ABB RAPID module: offs_inline.mod

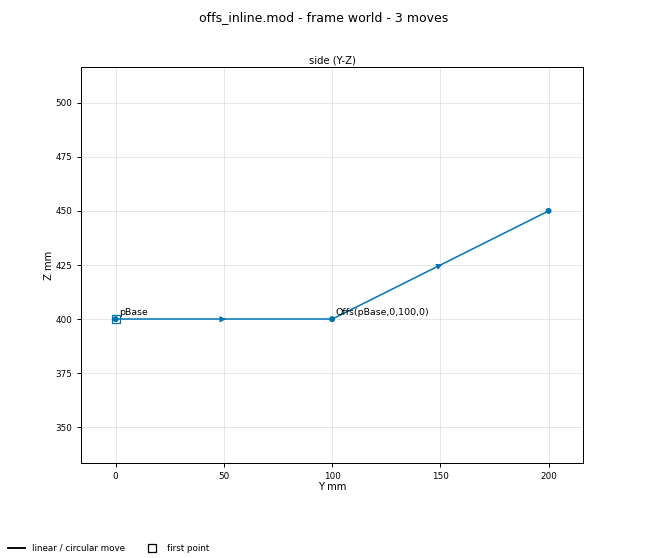
[picture p0: tool path of offs_inline.mod in frame world, 3 of 3 moves have a stored position in this frame; points joined in program order, loops and branches not executed]
MODULE OffsTest
  CONST robtarget pBase := [[500,0,400],[1,0,0,0],[0,0,0,0],[9E+09,9E+09,9E+09,9E+09,9E+09,9E+09]];

  PROC main()
    MoveL pBase, v100, fine, tool0;
    MoveL Offs(pBase, 0, 100, 0), v100, fine, tool0;
    MoveL Offs(pBase, 0, 200, 50), v100, z10, tool0;
  ENDPROC
ENDMODULE
